FUNCTION_BLOCK ABSTRACT FB_BaseDevice

VAR_INPUT
	name : WSTRING(255);
	location : WSTRING(255);
	description : WSTRING(255);
END_VAR

VAR
	monitoredDevice : FB_MonitoredDevice;
END_VAR

monitoredDevice.name := name;
monitoredDevice.location := location;
monitoredDevice.description := description;

METHOD FB_init : BOOL
VAR_INPUT
	bInitRetains : BOOL; // if TRUE, the retain variables are initialized (warm start / cold start)
	bInCopyCode : BOOL;  // if TRUE, the instance afterwards gets moved into the copy code (online change)
	name : WSTRING(255);
	location : WSTRING(255);
	description : WSTRING(255);
END_VAR
END_METHOD

END_FUNCTION_BLOCK

(* stored: Version 1.1.0.1, ProductVersion 3.1.4024.11
   POU FB_BaseDevice: Id {d7721b8f-bee1-4cfa-8b14-7db4e9e8b25c}, SpecialFunc None
   Method FB_init: Id {3a05c8df-e0c8-4643-ba2a-7fc74bd62ca9} *)
